// TIA Portal V19 export
DATA_BLOCK "Uhrzeit"   // DB8
// stored: AutoNumber false, InstanceOfName Uhrzeit_WSU, InstanceOfType FB
"Uhrzeit_WSU"
   // VAR RETAIN
   //    aktDatum : DTL;
   //    Time_to_on : Int;
   //    Time_to_off : Int;
   //    min_of_week : Int;
   //    BA_Uhr_Ein : Bool;
   //    BA_Uhr_Dauer : Bool;
   //    AZ_aktiv : Bool;
   //    ProfileWeek : Array[0..28] of Struct
   //       MinWeek : Int;
   //       State : Byte;
   //       resB : Byte;
   //    END_STRUCT;
   // END_VAR
BEGIN
END_DATA_BLOCK
